FUNCTION_BLOCK FB_simulatedpompdigout IMPLEMENTS ITF_pompdigout
VAR
	internalState:BOOL;
END_VAR

{warning 'Add method implementation '}
METHOD set : BOOL
VAR_INPUT
	state	: BOOL;
END_VAR
internalState := state;
END_METHOD

END_FUNCTION_BLOCK

(* stored: Version 1.1.0.1, ProductVersion 3.1.4026.8
   POU FB_simulatedpompdigout: Id {e7c545b7-e0f2-414e-8148-4f7973fdb8d3}, SpecialFunc None
   Method set: Id {24160de5-cbd3-4a03-9332-d573fcb15dc3} *)
